FUNCTION_BLOCK EL4102
VAR
	_io : EL4xx2_Data;
	{attribute addProperty Name "WcState"}
	_wcState : WcStateBase;
	{attribute addProperty Name "Info data"}
	_infoData : InfoDataAds;
END_VAR

PROPERTY IO : REFERENCE TO EL4xx2_Data
GET
IO REF= _io;
END_GET
END_PROPERTY

PROPERTY WcState : REFERENCE TO WcStateBase
GET
WcState REF= _wcState;
END_GET
END_PROPERTY

END_FUNCTION_BLOCK

(* stored: Version 1.1.0.1, ProductVersion 3.1.4024.9
   POU EL4102: Id {905e8189-ab39-0281-1745-a39ee4703fbd}, SpecialFunc None
   Property IO: Id {2f37dbc2-f8dd-0270-0fd3-5a5624900023}
   Get Get: Id {2d506a16-35b6-00f1-1704-fa74aaf5834c}
   Property WcState: Id {52c2cd25-8767-0a71-0e4e-4778baac438b}
   Get Get: Id {6a8e0245-0b46-0c74-145c-77790e5de75e} *)
